(* Schneider Machine Expert - Basic project sequential motor system for 3 motors, file version 2.7.0.0 *)
(* ProjectInformations: Name=New project *)

HARDWARE
  Cpu 0: TM221M16R/G
  EthernetConfiguration: NetworkName=M221, IpAllocationMode=FixedAddress, IpAddress=0.0.0.0, SubnetMask=0.0.0.0
  SerialLineConfiguration: Baud=Baud19200, Parity=ParityEven, DataBits=DataBits8, StopBits=StopBits1, PhysicalMedium=PhysicalMediumRs485, TransmissionMode=TransmissionModeModbusRtu, SlaveId=1, Addressing=SlaveAddressing
  MastTask: UsePeriodScanMode=false, PeriodScan=100
  FastTask: Period=255
  CpuBehavior: StartingMode=StartAsPreviousState, AutoSaveRamOnEeprom=true, WatchdogPeriod=250

SYMBOLS  (address, symbol, comment, settings)
  %M0       SEQQ_GOES_BRRR
  %TM0        [Preset=10, Base=OneSecond]
  %I0.0     STARTING
  %I0.1     STOP
  %Q0.0     MOTOR1
  %Q0.1     MOTOR2
  %Q0.2     MOTOR3

POU New POU
  (* SectionNumber=1 *)

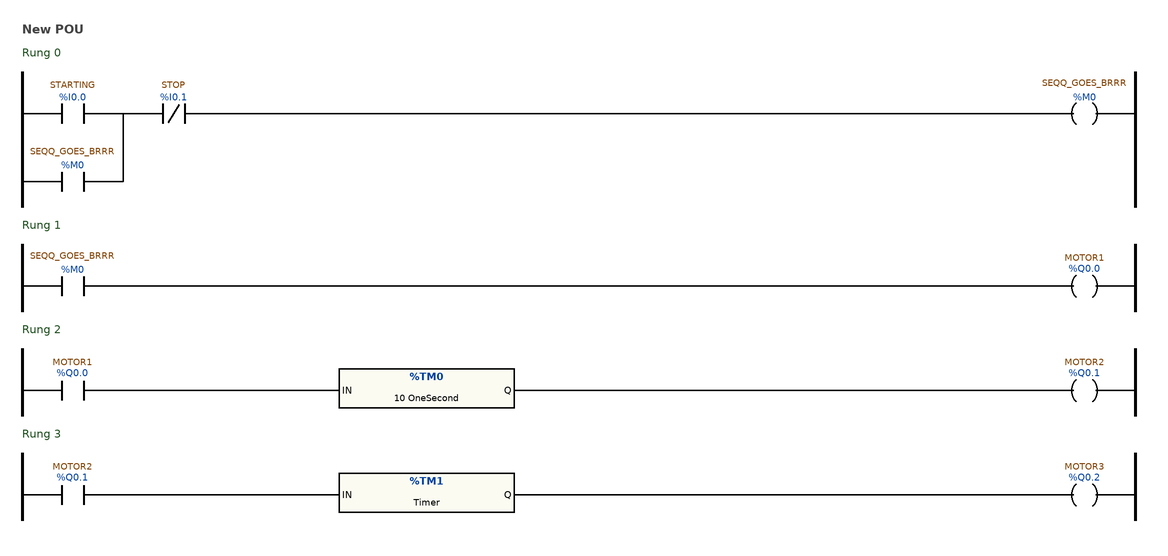

// Rung 0
  LD %I0.0                (* STARTING *)
  OR %M0                  (* SEQQ_GOES_BRRR *)
  ANDN %I0.1              (* STOP *)
  ST %M0                  (* SEQQ_GOES_BRRR *)
  // as ST:
  //   SEQQ_GOES_BRRR := (STARTING OR SEQQ_GOES_BRRR) AND NOT STOP;

// Rung 1
  LD %M0                  (* SEQQ_GOES_BRRR *)
  ST %Q0.0                (* MOTOR1 *)
  // as ST:
  //   MOTOR1 := SEQQ_GOES_BRRR;

// Rung 2
  BLK %TM0
  LD %Q0.0                (* MOTOR1 *)
  IN
  OUT_BLK
  LD Q
  ST %Q0.1                (* MOTOR2 *)
  END_BLK
  // as ST:
  //   %TM0(IN := MOTOR1);
  //   MOTOR2 := %TM0.Q;

// Rung 3
  BLK %TM1
  LD %Q0.1                (* MOTOR2 *)
  IN
  OUT_BLK
  LD Q
  ST %Q0.2                (* MOTOR3 *)
  END_BLK
  // as ST:
  //   %TM1(IN := MOTOR2);
  //   MOTOR3 := %TM1.Q;
